// TIA Portal V19 export
DATA_BLOCK "Alarms"   // DB95
// stored: MemoryReserve 100, Namespace Unit2.EM0
   VAR
      emAlarms { ExternalWritable := 'False'} : Array[0.._.Unit2_NO_OF_EMs] of "LAF_typeAlarms";
      errorNoReaction { ExternalWritable := 'False'} : Array[0..9] of Bool;   // Error without further impact / Error ohne weitere Auswirkungen
      errorAbort { ExternalWritable := 'False'} : Array[0..9] of Bool;   // Error which aborts the whole Unit / Error der ein abort in der Unit auslöst
      errorStop { ExternalWritable := 'False'} : Array[0..9] of Bool;   // Error which stops the whole Unit / Error der ein stop in der Unit auslöst
      warningNoReaction { ExternalWritable := 'False'} : Array[0..9] of Bool;   // Warning which could lead to a error / Warnung die zu einem Error führen kann
      warningHold { ExternalWritable := 'False'} : Array[0..9] of Bool;   // Warning which holds the whole Unit / Warnung die ein hold in der Unit auslöst
      warningSuspend { ExternalWritable := 'False'} : Array[0..9] of Bool;   // Warning which suspends the whole Unit / Warnung die ein suspend in der Unit auslöst
      information { ExternalWritable := 'False'} : Array[0..9] of Bool;   // Informations of the EM / Information des EM
      criteriaAnalysis { ExternalWritable := 'False'} : Array[0..9] of Bool;   // CriteriaAnalysis of the EM / Kriterienanalyse des EM
   END_VAR
BEGIN
   information[0] := false;
END_DATA_BLOCK
